SUBAPPLICATION InputOutputTesterBt_OPC_UA (* Tester *)
  (* Standard: 61499-2; Description: Copyright (c) 2023 Meisterschulen am Ostbahnhof This program and the accompanying materials are made available under the terms of the Eclipse Public License 2.0 which is available at https://www.eclipse.org/legal/epl-2.0/ SPDX-License-Identifier: EPL-2.0 *)
  (* Version 1.0, 2023-10-23, Franz Höpfinger, Meisterschulen am Ostbahnhof, initial API and implementation and/or initial documentation *)
  PACKAGE Meins::InputOutputTester::Button_OPC_UA;
  IMPORT Meins::InputOutputTester::Button_OPC_UA::SubStrings::I1_WRITE;
  IMPORT Meins::InputOutputTester::Button_OPC_UA::SubStrings::I2_WRITE;
  IMPORT Meins::InputOutputTester::Button_OPC_UA::SubStrings::I3_WRITE;
  IMPORT Meins::InputOutputTester::Button_OPC_UA::SubStrings::I4_WRITE;
  IMPORT Meins::InputOutputTester::Button_OPC_UA::SubStrings::I5_WRITE;
  IMPORT Meins::InputOutputTester::Button_OPC_UA::SubStrings::I6_WRITE;
  IMPORT Meins::InputOutputTester::Button_OPC_UA::SubStrings::I7_WRITE;
  IMPORT Meins::InputOutputTester::Button_OPC_UA::SubStrings::I8_WRITE;
  IMPORT Meins::InputOutputTester::Button_OPC_UA::SubStrings::Q01_READ;
  IMPORT Meins::InputOutputTester::Button_OPC_UA::SubStrings::Q01_WRITE;
  IMPORT Meins::InputOutputTester::Button_OPC_UA::SubStrings::Q02_READ;
  IMPORT Meins::InputOutputTester::Button_OPC_UA::SubStrings::Q02_WRITE;
  IMPORT Meins::InputOutputTester::Button_OPC_UA::SubStrings::Q03_READ;
  IMPORT Meins::InputOutputTester::Button_OPC_UA::SubStrings::Q03_WRITE;
  IMPORT Meins::InputOutputTester::Button_OPC_UA::SubStrings::Q04_READ;
  IMPORT Meins::InputOutputTester::Button_OPC_UA::SubStrings::Q04_WRITE;
  IMPORT Meins::InputOutputTester::Button_OPC_UA::SubStrings::Q05_READ;
  IMPORT Meins::InputOutputTester::Button_OPC_UA::SubStrings::Q05_WRITE;
  IMPORT Meins::InputOutputTester::Button_OPC_UA::SubStrings::Q06_READ;
  IMPORT Meins::InputOutputTester::Button_OPC_UA::SubStrings::Q06_WRITE;
  IMPORT Meins::InputOutputTester::Button_OPC_UA::SubStrings::Q07_READ;
  IMPORT Meins::InputOutputTester::Button_OPC_UA::SubStrings::Q07_WRITE;
  IMPORT Meins::InputOutputTester::Button_OPC_UA::SubStrings::Q08_READ;
  IMPORT Meins::InputOutputTester::Button_OPC_UA::SubStrings::Q08_WRITE;
  IMPORT Meins::InputOutputTester::Button_OPC_UA::SubStrings::Q09_READ;
  IMPORT Meins::InputOutputTester::Button_OPC_UA::SubStrings::Q09_WRITE;
  IMPORT Meins::InputOutputTester::Button_OPC_UA::SubStrings::Q10_READ;
  IMPORT Meins::InputOutputTester::Button_OPC_UA::SubStrings::Q10_WRITE;
  IMPORT Meins::InputOutputTester::Button_OPC_UA::SubStrings::Q11_READ;
  IMPORT Meins::InputOutputTester::Button_OPC_UA::SubStrings::Q11_WRITE;
  IMPORT Meins::InputOutputTester::Button_OPC_UA::SubStrings::Q12_READ;
  IMPORT Meins::InputOutputTester::Button_OPC_UA::SubStrings::Q12_WRITE;
  IMPORT Uebungen::const::UT::Tester::DefaultPool_Tester::Button_I01;
  IMPORT Uebungen::const::UT::Tester::DefaultPool_Tester::Button_I02;
  IMPORT Uebungen::const::UT::Tester::DefaultPool_Tester::Button_I03;
  IMPORT Uebungen::const::UT::Tester::DefaultPool_Tester::Button_I04;
  IMPORT Uebungen::const::UT::Tester::DefaultPool_Tester::Button_I05;
  IMPORT Uebungen::const::UT::Tester::DefaultPool_Tester::Button_I06;
  IMPORT Uebungen::const::UT::Tester::DefaultPool_Tester::Button_I07;
  IMPORT Uebungen::const::UT::Tester::DefaultPool_Tester::Button_I08;
  IMPORT Uebungen::const::UT::Tester::DefaultPool_Tester::Button_Q01;
  IMPORT Uebungen::const::UT::Tester::DefaultPool_Tester::Button_Q02;
  IMPORT Uebungen::const::UT::Tester::DefaultPool_Tester::Button_Q03;
  IMPORT Uebungen::const::UT::Tester::DefaultPool_Tester::Button_Q04;
  IMPORT Uebungen::const::UT::Tester::DefaultPool_Tester::Button_Q05;
  IMPORT Uebungen::const::UT::Tester::DefaultPool_Tester::Button_Q06;
  IMPORT Uebungen::const::UT::Tester::DefaultPool_Tester::Button_Q07;
  IMPORT Uebungen::const::UT::Tester::DefaultPool_Tester::Button_Q08;
  IMPORT Uebungen::const::UT::Tester::DefaultPool_Tester::Button_Q09;
  IMPORT Uebungen::const::UT::Tester::DefaultPool_Tester::Button_Q10;
  IMPORT Uebungen::const::UT::Tester::DefaultPool_Tester::Button_Q11;
  IMPORT Uebungen::const::UT::Tester::DefaultPool_Tester::Button_Q12;
  IMPORT logiBUS::io::DI::logiBUS_DI::Input_I1;
  IMPORT logiBUS::io::DI::logiBUS_DI::Input_I2;
  IMPORT logiBUS::io::DI::logiBUS_DI::Input_I3;
  IMPORT logiBUS::io::DI::logiBUS_DI::Input_I4;
  IMPORT logiBUS::io::DI::logiBUS_DI::Input_I5;
  IMPORT logiBUS::io::DI::logiBUS_DI::Input_I6;
  IMPORT logiBUS::io::DI::logiBUS_DI::Input_I7;
  IMPORT logiBUS::io::DI::logiBUS_DI::Input_I8;
  IMPORT logiBUS::io::DQ::logiBUS_DO::Output_Q1;
  IMPORT logiBUS::io::DQ::logiBUS_DO::Output_Q10;
  IMPORT logiBUS::io::DQ::logiBUS_DO::Output_Q11;
  IMPORT logiBUS::io::DQ::logiBUS_DO::Output_Q12;
  IMPORT logiBUS::io::DQ::logiBUS_DO::Output_Q2;
  IMPORT logiBUS::io::DQ::logiBUS_DO::Output_Q3;
  IMPORT logiBUS::io::DQ::logiBUS_DO::Output_Q4;
  IMPORT logiBUS::io::DQ::logiBUS_DO::Output_Q5;
  IMPORT logiBUS::io::DQ::logiBUS_DO::Output_Q6;
  IMPORT logiBUS::io::DQ::logiBUS_DO::Output_Q7;
  IMPORT logiBUS::io::DQ::logiBUS_DO::Output_Q8;
  IMPORT logiBUS::io::DQ::logiBUS_DO::Output_Q9;
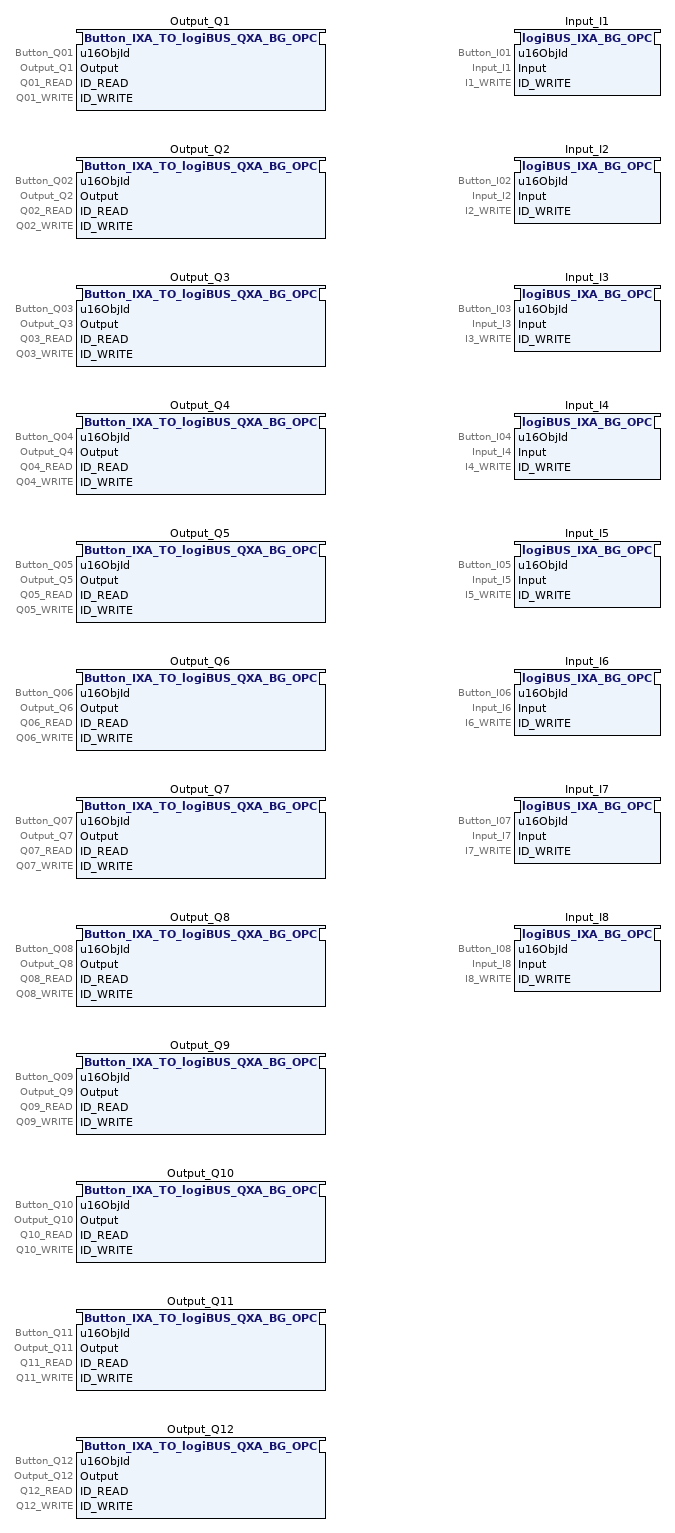
  SUBAPPS
    Input_I1 : MyLib::sys::logiBUS_IXA_BG_OPC(u16ObjId := Button_I01, Input := Input_I1, ID_WRITE := I1_WRITE);
    Input_I2 : MyLib::sys::logiBUS_IXA_BG_OPC(u16ObjId := Button_I02, Input := Input_I2, ID_WRITE := I2_WRITE);
    Input_I3 : MyLib::sys::logiBUS_IXA_BG_OPC(u16ObjId := Button_I03, Input := Input_I3, ID_WRITE := I3_WRITE);
    Input_I4 : MyLib::sys::logiBUS_IXA_BG_OPC(u16ObjId := Button_I04, Input := Input_I4, ID_WRITE := I4_WRITE);
    Input_I5 : MyLib::sys::logiBUS_IXA_BG_OPC(u16ObjId := Button_I05, Input := Input_I5, ID_WRITE := I5_WRITE);
    Input_I6 : MyLib::sys::logiBUS_IXA_BG_OPC(u16ObjId := Button_I06, Input := Input_I6, ID_WRITE := I6_WRITE);
    Input_I7 : MyLib::sys::logiBUS_IXA_BG_OPC(u16ObjId := Button_I07, Input := Input_I7, ID_WRITE := I7_WRITE);
    Input_I8 : MyLib::sys::logiBUS_IXA_BG_OPC(u16ObjId := Button_I08, Input := Input_I8, ID_WRITE := I8_WRITE);
    Output_Q1 : MyLib::sys::Button_IXA_TO_logiBUS_QXA_BG_OPC(u16ObjId := Button_Q01, Output := Output_Q1, ID_READ := Q01_READ, ID_WRITE := Q01_WRITE);
    Output_Q2 : MyLib::sys::Button_IXA_TO_logiBUS_QXA_BG_OPC(u16ObjId := Button_Q02, Output := Output_Q2, ID_READ := Q02_READ, ID_WRITE := Q02_WRITE);
    Output_Q3 : MyLib::sys::Button_IXA_TO_logiBUS_QXA_BG_OPC(u16ObjId := Button_Q03, Output := Output_Q3, ID_READ := Q03_READ, ID_WRITE := Q03_WRITE);
    Output_Q4 : MyLib::sys::Button_IXA_TO_logiBUS_QXA_BG_OPC(u16ObjId := Button_Q04, Output := Output_Q4, ID_READ := Q04_READ, ID_WRITE := Q04_WRITE);
    Output_Q5 : MyLib::sys::Button_IXA_TO_logiBUS_QXA_BG_OPC(u16ObjId := Button_Q05, Output := Output_Q5, ID_READ := Q05_READ, ID_WRITE := Q05_WRITE);
    Output_Q6 : MyLib::sys::Button_IXA_TO_logiBUS_QXA_BG_OPC(u16ObjId := Button_Q06, Output := Output_Q6, ID_READ := Q06_READ, ID_WRITE := Q06_WRITE);
    Output_Q7 : MyLib::sys::Button_IXA_TO_logiBUS_QXA_BG_OPC(u16ObjId := Button_Q07, Output := Output_Q7, ID_READ := Q07_READ, ID_WRITE := Q07_WRITE);
    Output_Q8 : MyLib::sys::Button_IXA_TO_logiBUS_QXA_BG_OPC(u16ObjId := Button_Q08, Output := Output_Q8, ID_READ := Q08_READ, ID_WRITE := Q08_WRITE);
    Output_Q9 : MyLib::sys::Button_IXA_TO_logiBUS_QXA_BG_OPC(u16ObjId := Button_Q09, Output := Output_Q9, ID_READ := Q09_READ, ID_WRITE := Q09_WRITE);
    Output_Q10 : MyLib::sys::Button_IXA_TO_logiBUS_QXA_BG_OPC(u16ObjId := Button_Q10, Output := Output_Q10, ID_READ := Q10_READ, ID_WRITE := Q10_WRITE);
    Output_Q11 : MyLib::sys::Button_IXA_TO_logiBUS_QXA_BG_OPC(u16ObjId := Button_Q11, Output := Output_Q11, ID_READ := Q11_READ, ID_WRITE := Q11_WRITE);
    Output_Q12 : MyLib::sys::Button_IXA_TO_logiBUS_QXA_BG_OPC(u16ObjId := Button_Q12, Output := Output_Q12, ID_READ := Q12_READ, ID_WRITE := Q12_WRITE);
  END_SUBAPPS
END_SUBAPPLICATION
